// TIA Portal V17 export
// export: Created 2024-09-02T12:50:04.7252641Z, ExportSetting WithDefaults, DisplayName Totally Integrated Automation Portal, DisplayVersion V17, DisplayName TIA Portal Openness, DisplayVersion V17, DisplayName TIA Portal Version Control Interface, DisplayVersion V17, DisplayName STEP 7 Professional, DisplayVersion V17, DisplayName STEP 7 Safety, DisplayVersion V17, DisplayName WinCC Professional, DisplayVersion V17
FUNCTION "SysFC_SQ_Mode" : Void   // FC180, LAD
TITLE = FC system / System FC
{ S7_Optimized_Access := 'TRUE' }
AUTHOR : OlegFuehrus
FAMILY : SK
NAME : SK
VERSION : 1.0
// stored: AutoNumber false, IsIECCheckEnabled false, SetENOAutomatically false, UDAEnableTagReadback false
   VAR_INPUT
      iFKT : Int;
      iTmsHalt : Bool;
   END_VAR
   VAR_IN_OUT
      ioMOP : G7_MOPPlus_V4;
   END_VAR
BEGIN

REGION Network 1: Status : Chain does not continue switching / Zustand: Kette schaltet nicht weiter
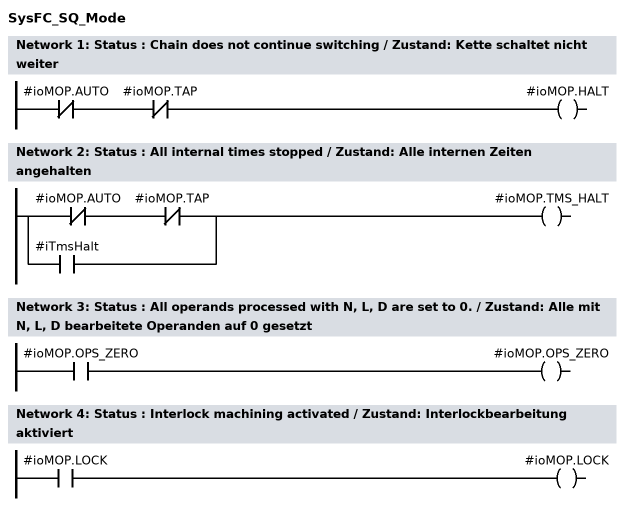
   RUNG wire#powerrail
      I_Contact( #ioMOP.AUTO )
      I_Contact( #ioMOP.TAP )
      Coil( #ioMOP.HALT )
   END_RUNG
   // the same network as SCL:
   #ioMOP.HALT := NOT #ioMOP.AUTO AND NOT #ioMOP.TAP;
END_REGION

REGION Network 2: Status : All internal times stopped / Zustand: Alle internen Zeiten angehalten
   RUNG wire#powerrail
      I_Contact( #ioMOP.AUTO )
      I_Contact( #ioMOP.TAP )
      wire#w1
      Coil( #ioMOP.TMS_HALT )
   END_RUNG
   RUNG wire#powerrail
      Contact( #iTmsHalt )
   END_RUNG wire#w1
   // the same network as SCL:
   #ioMOP.TMS_HALT := (NOT #ioMOP.AUTO AND NOT #ioMOP.TAP) OR #iTmsHalt;
END_REGION

REGION Network 3: Status : All operands processed with N, L, D are set to 0. / Zustand: Alle mit N, L, D bearbeitete Operanden auf 0 gesetzt
   RUNG wire#powerrail
      Contact( #ioMOP.OPS_ZERO )
      Coil( #ioMOP.OPS_ZERO )
   END_RUNG
   // the same network as SCL:
   #ioMOP.OPS_ZERO := #ioMOP.OPS_ZERO;
END_REGION

REGION Network 4: Status : Interlock machining activated / Zustand: Interlockbearbeitung aktiviert
   RUNG wire#powerrail
      Contact( #ioMOP.LOCK )
      Coil( #ioMOP.LOCK )
   END_RUNG
   // the same network as SCL:
   #ioMOP.LOCK := #ioMOP.LOCK;
END_REGION
END_FUNCTION
